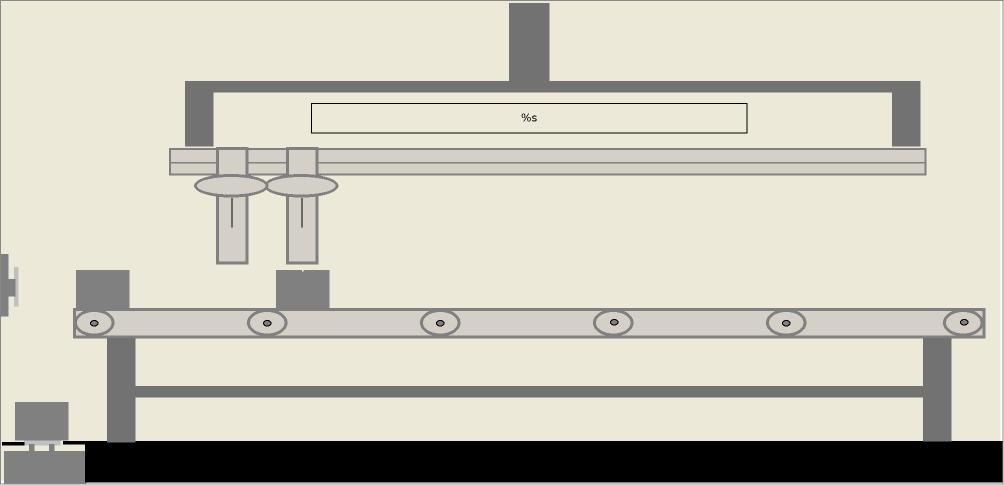
VISUALIZATION TC_FlyingSawPage  // 1004x485
    Rectangle (0,0 1000x480)
    RoundedRectangle (169,148 757x27)
    Rectangle (171,162 755x1)
    RoundedRectangle (73,308 912x30)
    Rectangle (4,451 82x32)
    RoundedRectangle (24,440 36x5)
        p2738717112: -(PRG_Simulation.nUp)
    Rectangle (85,441 917x41)
    Rectangle (63,441 34x3)
    Rectangle (29,444 5x8)
        p2773130477: -(PRG_Simulation.nUp)
    RoundedRectangle (49,444 5x8)
        p2773130477: -(PRG_Simulation.nUp)
    Rectangle (216,147 32x117), invisible if: PRG_Simulation.bMatkapInvisible
        p3560616238: Axis2.NcToPlc.ActPos/14.706
    Ellipse (194,174 74x23), invisible if: PRG_Simulation.bMatkapInvisible
        p2738717112: (Axis3.NcToPlc.ActPos)/15.38461538
        p3560616238: Axis2.NcToPlc.ActPos/14.706
    Line (232,227) (232,198), invisible if: PRG_Simulation.bMatkapInvisible
        p2738717112: (Axis3.NcToPlc.ActPos)/15.38461538
        p3560616238: Axis2.NcToPlc.ActPos/14.706
    Rectangle (76,270 53x38), invisible if: PRG_Simulation.bParca1Invisible
        p3560616238: Axis1.NcToPlc.ActPos/30
    Rectangle (276,270 53x38), invisible if: PRG_Simulation.bParca2Invisible2
        p3560616238: PRG_Simulation.fAxis1SimulationActPosX
    Rectangle (286,147 32x117), invisible if: PRG_Simulation.bMatkapInvisible2
        p3560616238: PRG_Simulation.fAxis2SimulationActPosX
    Ellipse (264,174 74x23), invisible if: PRG_Simulation.bMatkapInvisible2
        p2738717112: (Axis3.NcToPlc.ActPos)/15.38461538
        p3560616238: PRG_Simulation.fAxis2SimulationActPosX
    Rectangle (216,147 32x117), invisible if: PRG_Simulation.bMatkapInvisible3
        p3560616238: PRG_Simulation.fAxis2SimulationActPosX
    Ellipse (194,174 74x23), invisible if: PRG_Simulation.bMatkapInvisible3
        p2738717112: (Axis3.NcToPlc.ActPos)/15.38461538
        p3560616238: PRG_Simulation.fAxis2SimulationActPosX
    Line (232,227) (232,198), invisible if: PRG_Simulation.bMatkapInvisible3
        p2738717112: (Axis3.NcToPlc.ActPos)/15.38461538
        p3560616238: PRG_Simulation.fAxis2SimulationActPosX
    Rectangle (15,402 53x38), invisible if: PRG_Simulation.bParcaUpInvisible
        p3560616238: PRG_Simulation.nRight
        p2738717112: -(PRG_Simulation.nUp)
    Rectangle (2,442 22x3)
    Rectangle (0,254 8x62)
    Rectangle (14,267 4x39)
        p3560616238: PRG_Simulation.nRight
    Rectangle (8,279 7x17)
        p874137650: PRG_Simulation.nRight
    Rectangle (302,270 1x1), invisible if: PRG_Simulation.bParca2Invisible2
        p3560616238: PRG_Simulation.fAxis2SimulationActPosX
        p2773130477: PRG_Simulation.fAxis3SimulationActPosY
    Line (302,227) (302,198), invisible if: PRG_Simulation.bMatkapInvisible2
        p2738717112: (Axis3.NcToPlc.ActPos)/15.38461538
        p3560616238: PRG_Simulation.fAxis2SimulationActPosX
    Ellipse (74,309 40x27)
    Ellipse (247,309 40x27)
    Ellipse (420,309 40x27)
    Ellipse (593,309 40x27)
    Ellipse (766,309 40x27)
    Ellipse (943,309 40x27)
    Ellipse (90,320 8x6)
    Ellipse (263,320 8x6)
    Ellipse (436,320 8x6)
    Ellipse (610,319 8x6)
    Ellipse (782,320 8x6)
    Ellipse (960,319 8x6)
    Rectangle (107,338 28x104)
    Rectangle (923,338 28x103)
    Rectangle (131,386 794x11)
    Rectangle (185,81 735x11)
    Rectangle (892,90 28x56)
    Rectangle (185,90 28x56)
    Rectangle (509,3 40x79)
    Rectangle (311,103 436x30), "%s", text variable: PRG_FlyingSaw.sMsg
END_VISUALIZATION

(* stored: Version 1.1.0.1, ProductVersion 3.1.4022.12
   Visu TC_FlyingSawPage: Id {0684fa76-dc04-40e8-9748-e533d86b6ae9} *)
